KUKA KRL program: ps_res_c2.src, ps_res_c2.dat

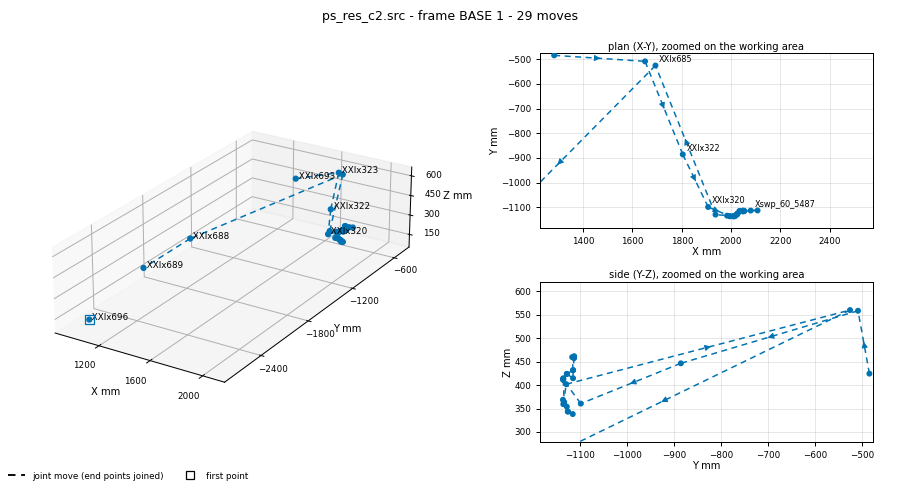
[picture p0: tool path of ps_res_c2.src in frame BASE 1, 29 of 34 moves have a stored position in this frame; points joined in program order, loops and branches not executed]
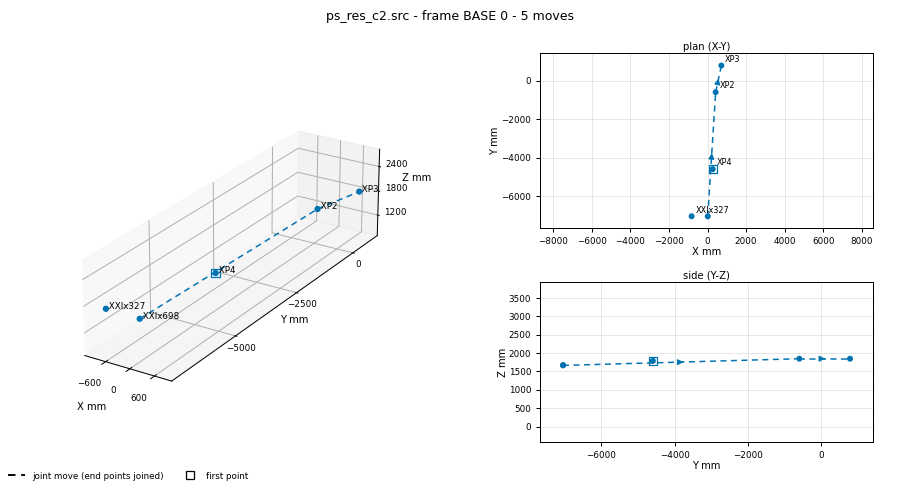
[picture p1: tool path of ps_res_c2.src in frame BASE 0, 5 of 34 moves have a stored position in this frame; points joined in program order, loops and branches not executed]
--- ps_res_c2.src ---
&ACCESS RVO1
&REL 115
&COMMENT Solda GUN C2 respot
&PARAM DISKPATH = KRC:\R1\Program
DEF ps_res_c2( )

;FOLD INI
;FOLD SPOTTECH INI
USERSPOT(#INIT)
;ENDFOLD (SPOTTECH INI)
;FOLD GRIPPERTECH INI
USER_GRP(0,DUMMY,DUMMY,GDEFAULT)
;ENDFOLD (GRIPPERTECH INI)
  ;FOLD USER INI
    ;Make your modifications here

  ;ENDFOLD (USER INI)
;ENDFOLD (INI)

; Caracterização dos meios de produção:
; Versão Atual:
; 08/06/2013 12:00 Name: P13.050-R1 CHANGES: Solda respot Actros
; Gun C2 (F2 6640 0018 997)

chk_w3_wechs_ok ( )              ; CHECK C2

if MaxStandMenge (2) then
 MaxStandmengeErreicht (2)
endif

IF (NOT(GHOST())) THEN
if Elektrodenwechsel (2) then
 e_fraes3 ()
endif
ENDIF

;FOLD OUT 3348 'Fora area GEOBOX' State=FALSE ;%{PE}%R 8.2.20,%MKUKATPBASIS,%COUT,%VOUTX,%P 2:3348, 3:Fora area GEOBOX, 5:FALSE, 6:
$OUT[3348]=FALSE
;ENDFOLD

;FOLD PTP P4 CONT Vel=100 % PDAT40 Tool[3]:GUN C2 Base[0];%{PE}%R 8.2.20,%MKUKATPBASIS,%CMOVE,%VPTP,%P 1:PTP, 2:P4, 3:C_DIS, 5:100, 7:PDAT40
$BWDSTART=FALSE
PDAT_ACT=PPDAT40
FDAT_ACT=FP4
BAS(#PTP_PARAMS,100)
PTP XP4 C_DIS
;ENDFOLD

;FOLD Collision.Monitoring_3_On ;%{PE}%MKUKATPUSER
COLLSTOP( 3, 1 ) ;Interrupt-Controlled
;ENDFOLD

;FOLD PTP Xlx696 CONT Vel=100 % PDAT23 Tool[3]:GUN C2 Base[0];%{PE}%R 8.2.20,%MKUKATPBASIS,%CMOVE,%VPTP,%P 1:PTP, 2:Xlx696, 3:C_DIS, 5:100, 7:PDAT23
$BWDSTART=FALSE
PDAT_ACT=PPDAT23
FDAT_ACT=FXlx696
BAS(#PTP_PARAMS,100)
PTP XXlx696 C_DIS
;ENDFOLD

;FOLD Collision.Monitoring_5_On ;%{PE}%MKUKATPUSER
COLLSTOP( 5, 1 ) ;not Interrupt-Controlled
;ENDFOLD

;FOLD PTP Xlx327 CONT Vel=100 % P_OLP22 Tool[3]:GUN C2 Base[0];%{PE}%R 8.2.20,%MKUKATPBASIS,%CMOVE,%VPTP,%P 1:PTP, 2:Xlx327, 3:C_DIS, 5:100, 7:P_OLP22
$BWDSTART=FALSE
PDAT_ACT=PP_OLP22
FDAT_ACT=FXlx327
BAS(#PTP_PARAMS,100)
PTP XXlx327 C_DIS
;ENDFOLD

;LIGA INTERTRAVAMENTO 15 C/R5
;FOLD Collision.Monitoring_AREA_9_On ;%{PE}%MKUKATPUSER
COLLSTOP( 15, 1 ) ;not Interrupt-Controlled
;ENDFOLD

;FOLD PTP Xlx693 CONT Vel=100 % PDAT20 Tool[3]:GUN C2 Base[0];%{PE}%R 8.2.20,%MKUKATPBASIS,%CMOVE,%VPTP,%P 1:PTP, 2:Xlx693, 3:C_DIS, 5:100, 7:PDAT20
$BWDSTART=FALSE
PDAT_ACT=PPDAT20
FDAT_ACT=FXlx693
BAS(#PTP_PARAMS,100)
PTP XXlx693 C_DIS
;ENDFOLD
;FOLD PTP Xlx323 CONT Vel=100 % P_OLP3 Tool[3]:GUN C2 Base[0];%{PE}%R 8.2.19,%MKUKATPBASIS,%CMOVE,%VPTP,%P 1:PTP, 2:Xlx323, 3:C_DIS, 5:100, 7:P_OLP3
$BWDSTART=FALSE
PDAT_ACT=PP_OLP3
FDAT_ACT=FXlx323
BAS(#PTP_PARAMS,100)
PTP XXlx323 C_DIS
;ENDFOLD
;FOLD PTP Xlx322 CONT Vel=100 % P_OLP4 Tool[3]:GUN C2 Base[0];%{PE}%R 8.2.19,%MKUKATPBASIS,%CMOVE,%VPTP,%P 1:PTP, 2:Xlx322, 3:C_DIS, 5:100, 7:P_OLP4
$BWDSTART=FALSE
PDAT_ACT=PP_OLP4
FDAT_ACT=FXlx322
BAS(#PTP_PARAMS,100)
PTP XXlx322 C_DIS
;ENDFOLD
;FOLD PTP Xlx320 CONT Vel=100 % P_OLP6 Tool[3]:GUN C2 Base[0];%{PE}%R 8.2.19,%MKUKATPBASIS,%CMOVE,%VPTP,%P 1:PTP, 2:Xlx320, 3:C_DIS, 5:100, 7:P_OLP6
$BWDSTART=FALSE
PDAT_ACT=PP_OLP6
FDAT_ACT=FXlx320
BAS(#PTP_PARAMS,100)
PTP XXlx320 C_DIS
;ENDFOLD
;FOLD PTP Xlx669 CONT Vel=100 % PDAT26 Tool[3]:GUN C2 Base[0];%{PE}%R 8.2.20,%MKUKATPBASIS,%CMOVE,%VPTP,%P 1:PTP, 2:Xlx669, 3:C_DIS, 5:100, 7:PDAT26
$BWDSTART=FALSE
PDAT_ACT=PPDAT26
FDAT_ACT=FXlx669
BAS(#PTP_PARAMS,100)
PTP XXlx669 C_DIS
;ENDFOLD
;FOLD PTP Xlx670 CONT Vel=80 % PDAT27 Tool[3]:GUN C2 Base[0];%{PE}%R 8.2.20,%MKUKATPBASIS,%CMOVE,%VPTP,%P 1:PTP, 2:Xlx670, 3:C_DIS, 5:80, 7:PDAT27
$BWDSTART=FALSE
PDAT_ACT=PPDAT27
FDAT_ACT=FXlx670
BAS(#PTP_PARAMS,80)
PTP XXlx670 C_DIS
;ENDFOLD
;FOLD PTP Xlx672 CONT Vel=80 % PDAT7 Tool[3]:GUN C2 Base[0];%{PE}%R 8.2.20,%MKUKATPBASIS,%CMOVE,%VPTP,%P 1:PTP, 2:Xlx672, 3:C_DIS, 5:80, 7:PDAT7
$BWDSTART=FALSE
PDAT_ACT=PPDAT7
FDAT_ACT=FXlx672
BAS(#PTP_PARAMS,80)
PTP XXlx672 C_DIS
;ENDFOLD

;FOLD ; swp_60_5491;%{PE}%R 8.2.20,%MKUKATPBASIS,%CCOMMENT,%VNORMAL,%P 2:swp_60_5491
;ENDFOLD
;FOLD PTP swp_60_5491 P_OLP7 SPOT Gun=2 RETR CLS PgNo1=61 ACTIVE=1 Tool[3]:GUN C2 Base[1]:Actros;%{PE}%R 8.2.2,%MKUKATPSPOT,%CSPOT,%VPTP,%P 1:PTP, 2:swp_60_5491, 3:, 5:100, 7:P_OLP7, 10:2, 12:#FIRST, 14:#CLO, 16:61, 18:1, 20:1, 22:0, 24:1, 25:S_OLP1
$BWDSTART=FALSE
PDAT_ACT=PP_OLP7
FDAT_ACT=Fswp_60_5491
BAS(#PTP_PARAMS,PP_OLP7.VEL)
S_ACT.GUN=2
S_ACT.PAIR=SDEFAULT.PAIR
S_ACT.RETR=#CLO
S_ACT.CLO_TM=1
S_ACT.PGNO1=61
S_ACT.PGNO2=SDEFAULT.PGNO2
S_ACT.PRESS1=SDEFAULT.PRESS1
S_ACT.PRESS2=SDEFAULT.PRESS2
S_READY=FALSE
PTP Xswp_60_5491
USERSPOT(#SPOT, S_ACT)
WAIT FOR S_READY
;ENDFOLD

;FOLD ; swp_60_5489;%{PE}%R 8.2.20,%MKUKATPBASIS,%CCOMMENT,%VNORMAL,%P 2:swp_60_5489
;ENDFOLD
;FOLD PTP swp_60_5489 P_OLP8 SPOT Gun=2 RETR CLS PgNo1=62 ACTIVE=1 Tool[3]:GUN C2 Base[1]:Actros;%{PE}%R 8.2.2,%MKUKATPSPOT,%CSPOT,%VPTP,%P 1:PTP, 2:swp_60_5489, 3:, 5:100, 7:P_OLP8, 10:2, 12:#FIRST, 14:#CLO, 16:62, 18:1, 20:1, 22:0, 24:1, 25:S_OLP2
$BWDSTART=FALSE
PDAT_ACT=PP_OLP8
FDAT_ACT=Fswp_60_5489
BAS(#PTP_PARAMS,PP_OLP8.VEL)
S_ACT.GUN=2
S_ACT.PAIR=SDEFAULT.PAIR
S_ACT.RETR=#CLO
S_ACT.CLO_TM=1
S_ACT.PGNO1=62
S_ACT.PGNO2=SDEFAULT.PGNO2
S_ACT.PRESS1=SDEFAULT.PRESS1
S_ACT.PRESS2=SDEFAULT.PRESS2
S_READY=FALSE
PTP Xswp_60_5489
USERSPOT(#SPOT, S_ACT)
WAIT FOR S_READY
;ENDFOLD

;FOLD PTP Xlx674 CONT Vel=100 % PDAT29 Tool[3]:GUN C2 Base[0];%{PE}%R 8.2.20,%MKUKATPBASIS,%CMOVE,%VPTP,%P 1:PTP, 2:Xlx674, 3:C_DIS, 5:100, 7:PDAT29
$BWDSTART=FALSE
PDAT_ACT=PPDAT29
FDAT_ACT=FXlx674
BAS(#PTP_PARAMS,100)
PTP XXlx674 C_DIS
;ENDFOLD

;FOLD ; swp_60_5487;%{PE}%R 8.2.20,%MKUKATPBASIS,%CCOMMENT,%VNORMAL,%P 2:swp_60_5487
;ENDFOLD
;FOLD PTP swp_60_5487 P_OLP9 SPOT Gun=2 RETR CLS PgNo1=63 ACTIVE=1 Tool[3]:GUN C2 Base[1]:Actros;%{PE}%R 8.2.2,%MKUKATPSPOT,%CSPOT,%VPTP,%P 1:PTP, 2:swp_60_5487, 3:, 5:100, 7:P_OLP9, 10:2, 12:#FIRST, 14:#CLO, 16:63, 18:1, 20:1, 22:0, 24:1, 25:S_OLP3
$BWDSTART=FALSE
PDAT_ACT=PP_OLP9
FDAT_ACT=Fswp_60_5487
BAS(#PTP_PARAMS,PP_OLP9.VEL)
S_ACT.GUN=2
S_ACT.PAIR=SDEFAULT.PAIR
S_ACT.RETR=#CLO
S_ACT.CLO_TM=1
S_ACT.PGNO1=63
S_ACT.PGNO2=SDEFAULT.PGNO2
S_ACT.PRESS1=SDEFAULT.PRESS1
S_ACT.PRESS2=SDEFAULT.PRESS2
S_READY=FALSE
PTP Xswp_60_5487
USERSPOT(#SPOT, S_ACT)
WAIT FOR S_READY
;ENDFOLD

;FOLD ; swp_60_5485;%{PE}%R 8.2.20,%MKUKATPBASIS,%CCOMMENT,%VNORMAL,%P 2:swp_60_5485
;ENDFOLD
;FOLD PTP swp_60_5485 P_OLP10 SPOT Gun=2 RETR CLS PgNo1=64 ACTIVE=1 Tool[3]:GUN C2 Base[1]:Actros;%{PE}%R 8.2.2,%MKUKATPSPOT,%CSPOT,%VPTP,%P 1:PTP, 2:swp_60_5485, 3:, 5:100, 7:P_OLP10, 10:2, 12:#FIRST, 14:#CLO, 16:64, 18:1, 20:1, 22:0, 24:1, 25:S_OLP4
$BWDSTART=FALSE
PDAT_ACT=PP_OLP10
FDAT_ACT=Fswp_60_5485
BAS(#PTP_PARAMS,PP_OLP10.VEL)
S_ACT.GUN=2
S_ACT.PAIR=SDEFAULT.PAIR
S_ACT.RETR=#CLO
S_ACT.CLO_TM=1
S_ACT.PGNO1=64
S_ACT.PGNO2=SDEFAULT.PGNO2
S_ACT.PRESS1=SDEFAULT.PRESS1
S_ACT.PRESS2=SDEFAULT.PRESS2
S_READY=FALSE
PTP Xswp_60_5485
USERSPOT(#SPOT, S_ACT)
WAIT FOR S_READY
;ENDFOLD

;FOLD PTP Xlx328 CONT Vel=100 % PDAT30 Tool[3]:GUN C2 Base[0];%{PE}%R 8.2.20,%MKUKATPBASIS,%CMOVE,%VPTP,%P 1:PTP, 2:Xlx328, 3:C_DIS, 5:100, 7:PDAT30
$BWDSTART=FALSE
PDAT_ACT=PPDAT30
FDAT_ACT=FXlx328
BAS(#PTP_PARAMS,100)
PTP XXlx328 C_DIS
;ENDFOLD
;FOLD PTP Xlx329 CONT Vel=100 % P_OLP12 Tool[3]:GUN C2 Base[0];%{PE}%R 8.2.19,%MKUKATPBASIS,%CMOVE,%VPTP,%P 1:PTP, 2:Xlx329, 3:C_DIS, 5:100, 7:P_OLP12
$BWDSTART=FALSE
PDAT_ACT=PP_OLP12
FDAT_ACT=FXlx329
BAS(#PTP_PARAMS,100)
PTP XXlx329 C_DIS
;ENDFOLD
;FOLD PTP Xlx330 CONT Vel=100 % P_OLP13 Tool[3]:GUN C2 Base[0];%{PE}%R 8.2.19,%MKUKATPBASIS,%CMOVE,%VPTP,%P 1:PTP, 2:Xlx330, 3:C_DIS, 5:100, 7:P_OLP13
$BWDSTART=FALSE
PDAT_ACT=PP_OLP13
FDAT_ACT=FXlx330
BAS(#PTP_PARAMS,100)
PTP XXlx330 C_DIS
;ENDFOLD
;FOLD PTP Xlx675 Vel=80 % PDAT31 Tool[3]:GUN C2 Base[1]:Actros;%{PE}%R 8.2.20,%MKUKATPBASIS,%CMOVE,%VPTP,%P 1:PTP, 2:Xlx675, 3:, 5:80, 7:PDAT31
$BWDSTART=FALSE
PDAT_ACT=PPDAT31
FDAT_ACT=FXlx675
BAS(#PTP_PARAMS,80)
PTP XXlx675
;ENDFOLD
;FOLD PTP Xlx676 CONT Vel=100 % PDAT32 Tool[3]:GUN C2 Base[0];%{PE}%R 8.2.20,%MKUKATPBASIS,%CMOVE,%VPTP,%P 1:PTP, 2:Xlx676, 3:C_DIS, 5:100, 7:PDAT32
$BWDSTART=FALSE
PDAT_ACT=PPDAT32
FDAT_ACT=FXlx676
BAS(#PTP_PARAMS,100)
PTP XXlx676 C_DIS
;ENDFOLD
;FOLD PTP Xlx678 CONT Vel=100 % PDAT33 Tool[3]:GUN C2 Base[0];%{PE}%R 8.2.20,%MKUKATPBASIS,%CMOVE,%VPTP,%P 1:PTP, 2:Xlx678, 3:C_DIS, 5:100, 7:PDAT33
$BWDSTART=FALSE
PDAT_ACT=PPDAT33
FDAT_ACT=FXlx678
BAS(#PTP_PARAMS,100)
PTP XXlx678 C_DIS
;ENDFOLD
;FOLD PTP Xlx679 Vel=80 % PDAT34 Tool[3]:GUN C2 Base[1]:Actros;%{PE}%R 8.2.20,%MKUKATPBASIS,%CMOVE,%VPTP,%P 1:PTP, 2:Xlx679, 3:, 5:80, 7:PDAT34
$BWDSTART=FALSE
PDAT_ACT=PPDAT34
FDAT_ACT=FXlx679
BAS(#PTP_PARAMS,80)
PTP XXlx679
;ENDFOLD
;FOLD PTP Xlx680 CONT Vel=100 % PDAT35 Tool[3]:GUN C2 Base[0];%{PE}%R 8.2.20,%MKUKATPBASIS,%CMOVE,%VPTP,%P 1:PTP, 2:Xlx680, 3:C_DIS, 5:100, 7:PDAT35
$BWDSTART=FALSE
PDAT_ACT=PPDAT35
FDAT_ACT=FXlx680
BAS(#PTP_PARAMS,100)
PTP XXlx680 C_DIS
;ENDFOLD
;FOLD PTP Xlx682 CONT Vel=100 % PDAT10 Tool[3]:GUN C2 Base[0];%{PE}%R 8.2.19,%MKUKATPBASIS,%CMOVE,%VPTP,%P 1:PTP, 2:Xlx682, 3:C_DIS, 5:100, 7:PDAT10
$BWDSTART=FALSE
PDAT_ACT=PPDAT10
FDAT_ACT=FXlx682
BAS(#PTP_PARAMS,100)
PTP XXlx682 C_DIS
;ENDFOLD

;FOLD ; swp_60_5493;%{PE}%R 8.2.20,%MKUKATPBASIS,%CCOMMENT,%VNORMAL,%P 2:swp_60_5493
;ENDFOLD
;FOLD PTP swp_60_5493 P_OLP14 SPOT Gun=2 RETR CLS PgNo1=65 ACTIVE=1 Tool[3]:GUN C2 Base[1]:Actros;%{PE}%R 8.2.2,%MKUKATPSPOT,%CSPOT,%VPTP,%P 1:PTP, 2:swp_60_5493, 3:, 5:100, 7:P_OLP14, 10:2, 12:#FIRST, 14:#CLO, 16:65, 18:1, 20:1, 22:0, 24:1, 25:S_OLP5
$BWDSTART=FALSE
PDAT_ACT=PP_OLP14
FDAT_ACT=Fswp_60_5493
BAS(#PTP_PARAMS,PP_OLP14.VEL)
S_ACT.GUN=2
S_ACT.PAIR=SDEFAULT.PAIR
S_ACT.RETR=#CLO
S_ACT.CLO_TM=1
S_ACT.PGNO1=65
S_ACT.PGNO2=SDEFAULT.PGNO2
S_ACT.PRESS1=SDEFAULT.PRESS1
S_ACT.PRESS2=SDEFAULT.PRESS2
S_READY=FALSE
PTP Xswp_60_5493
USERSPOT(#SPOT, S_ACT)
WAIT FOR S_READY
;ENDFOLD

;FOLD PTP Xlx331 CONT Vel=100 % P_OLP15 Tool[3]:GUN C2 Base[0];%{PE}%R 8.2.19,%MKUKATPBASIS,%CMOVE,%VPTP,%P 1:PTP, 2:Xlx331, 3:C_DIS, 5:100, 7:P_OLP15
$BWDSTART=FALSE
PDAT_ACT=PP_OLP15
FDAT_ACT=FXlx331
BAS(#PTP_PARAMS,100)
PTP XXlx331 C_DIS
;ENDFOLD
;FOLD PTP Xlx332 Vel=80 % P_OLP16 Tool[3]:GUN C2 Base[1]:Actros;%{PE}%R 8.2.20,%MKUKATPBASIS,%CMOVE,%VPTP,%P 1:PTP, 2:Xlx332, 3:, 5:80, 7:P_OLP16
$BWDSTART=FALSE
PDAT_ACT=PP_OLP16
FDAT_ACT=FXlx332
BAS(#PTP_PARAMS,80)
PTP XXlx332
;ENDFOLD
;FOLD PTP Xlx334 CONT Vel=100 % PDAT36 Tool[3]:GUN C2 Base[0];%{PE}%R 8.2.20,%MKUKATPBASIS,%CMOVE,%VPTP,%P 1:PTP, 2:Xlx334, 3:C_DIS, 5:100, 7:PDAT36
$BWDSTART=FALSE
PDAT_ACT=PPDAT36
FDAT_ACT=FXlx334
BAS(#PTP_PARAMS,100)
PTP XXlx334 C_DIS
;ENDFOLD
;FOLD PTP Xlx685 CONT Vel=100 % PDAT12 Tool[3]:GUN C2 Base[0];%{PE}%R 8.2.20,%MKUKATPBASIS,%CMOVE,%VPTP,%P 1:PTP, 2:Xlx685, 3:C_DIS, 5:100, 7:PDAT12
$BWDSTART=FALSE
PDAT_ACT=PPDAT12
FDAT_ACT=FXlx685
BAS(#PTP_PARAMS,100)
PTP XXlx685 C_DIS
;ENDFOLD
;FOLD PTP Xlx688 CONT Vel=100 % PDAT15 Tool[3]:GUN C2 Base[0];%{PE}%R 8.2.19,%MKUKATPBASIS,%CMOVE,%VPTP,%P 1:PTP, 2:Xlx688, 3:C_DIS, 5:100, 7:PDAT15
$BWDSTART=FALSE
PDAT_ACT=PPDAT15
FDAT_ACT=FXlx688
BAS(#PTP_PARAMS,100)
PTP XXlx688 C_DIS
;ENDFOLD
;FOLD PTP Xlx689 Vel=100 % PDAT16 Tool[3]:GUN C2 Base[1]:Actros;%{PE}%R 8.2.20,%MKUKATPBASIS,%CMOVE,%VPTP,%P 1:PTP, 2:Xlx689, 3:, 5:100, 7:PDAT16
$BWDSTART=FALSE
PDAT_ACT=PPDAT16
FDAT_ACT=FXlx689
BAS(#PTP_PARAMS,100)
PTP XXlx689
;ENDFOLD

;FOLD Collision.Monitoring_5_Off . ;%{PE}%MKUKATPUSER
COLLSTOP( 5, 2+0 )
;ENDFOLD

;DESLIGA INTERTRAVAMENTO 15 C/R5
;FOLD Collision.Monitoring_AREA_9_Off . ;%{PE}%MKUKATPUSER
COLLSTOP( 15, 2+0 )
;ENDFOLD

;FOLD PTP Xlx698 Vel=100 % PDAT25 Tool[3]:GUN C2 Base[0];%{PE}%R 8.2.20,%MKUKATPBASIS,%CMOVE,%VPTP,%P 1:PTP, 2:Xlx698, 3:, 5:100, 7:PDAT25
$BWDSTART=FALSE
PDAT_ACT=PPDAT25
FDAT_ACT=FXlx698
BAS(#PTP_PARAMS,100)
PTP XXlx698
;ENDFOLD

;FOLD Collision.Monitoring_3_On ;%{PE}%MKUKATPUSER
COLLSTOP( 3, 1 ) ;Interrupt-Controlled
;ENDFOLD
;FOLD OUT 3348 'Fora area GEOBOX' State=TRUE ;%{PE}%R 8.2.20,%MKUKATPBASIS,%COUT,%VOUTX,%P 2:3348, 3:Fora area GEOBOX, 5:TRUE, 6:
$OUT[3348]=TRUE
;ENDFOLD
;FOLD PULSE 3407 'RESPOT concluido' State=TRUE Time=2 sec;%{PE}%R 8.2.20,%MKUKATPBASIS,%COUT,%VPULSE,%P 2:3407, 3:RESPOT concluido, 5:TRUE, 6:, 8:2
PULSE($OUT[3407], TRUE,2)
;ENDFOLD
end_weld_RESPOT()             ; BIT FIM DE SOLDA RESPOT

;FOLD PTP P2 CONT Vel=100 % PDAT38 Tool[3]:GUN C2 Base[0];%{PE}%R 8.2.20,%MKUKATPBASIS,%CMOVE,%VPTP,%P 1:PTP, 2:P2, 3:C_DIS, 5:100, 7:PDAT38
$BWDSTART=FALSE
PDAT_ACT=PPDAT38
FDAT_ACT=FP2
BAS(#PTP_PARAMS,100)
PTP XP2 C_DIS
;ENDFOLD
;FOLD PTP P3 CONT Vel=100 % PDAT39 Tool[3]:GUN C2 Base[0];%{PE}%R 8.2.20,%MKUKATPBASIS,%CMOVE,%VPTP,%P 1:PTP, 2:P3, 3:C_DIS, 5:100, 7:PDAT39
$BWDSTART=FALSE
PDAT_ACT=PPDAT39
FDAT_ACT=FP3
BAS(#PTP_PARAMS,100)
PTP XP3 C_DIS
;ENDFOLD

IF (NOT(GHOST())) THEN
if FraesAnf (2) then
 e_fraes3 ()
endif
ENDIF

END

--- ps_res_c2.dat ---
&ACCESS RVO1
&REL 115
&COMMENT Solda GUN C2 respot
&PARAM DISKPATH = KRC:\R1\Program
DEFDAT  ps_res_c2
;FOLD EXTERNAL DECLARATIONS;%{PE}%MKUKATPBASIS,%CEXT,%VCOMMON,%P
;FOLD GRIPPERTECH EXT
EXT  H50 (INT  :IN,INT  :IN,INT  :IN,GRP_TYP  :IN )
;ENDFOLD (GRIPPERTECH EXT)
;FOLD SPOTTECH EXT
EXT  USERSPOT (S_COMMAND  :IN,SPOT_TYPE  :IN )
;ENDFOLD (SPOTTECH EXT)
;FOLD BASISTECH EXT;%{PE}%MKUKATPBASIS,%CEXT,%VEXT,%P
EXT  BAS (BAS_COMMAND  :IN,REAL  :IN )
DECL INT SUCCESS
;ENDFOLD (BASISTECH EXT)
;FOLD USER EXT;%{E}%MKUKATPUSER,%CEXT,%VEXT,%P
;Make your modifications here

;ENDFOLD (USER EXT)
;ENDFOLD (EXTERNAL DECLARATIONS)

;# ============ START PATH : swp_p13050r1_l_res_c2 =============
DECL PDAT PP_OLP3={VEL 100.0,ACC 100.0,APO_DIST 100.0,APO_MODE #CDIS}
DECL PDAT PP_OLP4={VEL 100.0,ACC 100.0,APO_DIST 100.0,APO_MODE #CDIS}
DECL PDAT PP_OLP6={VEL 100.0,ACC 100.0,APO_DIST 100.0,APO_MODE #CDIS}
DECL FDAT Fswp_60_5491={TOOL_NO 3,BASE_NO 1,IPO_FRAME #BASE,POINT2[] " "}
DECL PDAT PP_OLP7={VEL 100.0,ACC 100.0,APO_DIST 0.0}
DECL SPOT_TYPE SS_OLP1={GUN 1,PAIR #FIRST,RETR #CLO,CLO_TM 0,PGNO1 1,PRESS1 1.0,PGNO2 0,PRESS2 0.0}
DECL E6POS Xswp_60_5491={X 2034.40295,Y -1115.71399,Z 414.519287,A -0.537424684,B 7.66125584,C -86.3613815,S 2,T 2,E1 -7394.22998,E2 0.0,E3 0.0,E4 0.0,E5 0.0,E6 0.0}
DECL FDAT Fswp_60_5489={TOOL_NO 3,BASE_NO 1,IPO_FRAME #BASE,POINT2[] " "}
DECL PDAT PP_OLP8={VEL 100.0,ACC 100.0,APO_DIST 0.0}
DECL SPOT_TYPE SS_OLP2={GUN 1,PAIR #FIRST,RETR #CLO,CLO_TM 0,PGNO1 1,PRESS1 1.0,PGNO2 0,PRESS2 0.0}
DECL E6POS Xswp_60_5489={X 2053.09009,Y -1115.62305,Z 431.705597,A 0.718700528,B 7.58153105,C -86.2006226,S 2,T 2,E1 -7394.23096,E2 0.0,E3 0.0,E4 0.0,E5 0.0,E6 0.0}
DECL FDAT Fswp_60_5487={TOOL_NO 3,BASE_NO 1,IPO_FRAME #BASE,POINT2[] " "}
DECL PDAT PP_OLP9={VEL 100.0,ACC 100.0,APO_DIST 0.0}
DECL SPOT_TYPE SS_OLP3={GUN 1,PAIR #FIRST,RETR #CLO,CLO_TM 0,PGNO1 1,PRESS1 1.0,PGNO2 0,PRESS2 0.0}
DECL E6POS Xswp_60_5487={X 2079.30493,Y -1113.76294,Z 457.208313,A 0.301905006,B 1.24084997,C -86.230957,S 2,T 2,E1 -7394.229,E2 0.0,E3 0.0,E4 0.0,E5 0.0,E6 0.0}
DECL FDAT Fswp_60_5485={TOOL_NO 3,BASE_NO 1,IPO_FRAME #BASE,POINT2[] " "}
DECL PDAT PP_OLP10={VEL 100.0,ACC 100.0,APO_DIST 0.0}
DECL SPOT_TYPE SS_OLP4={GUN 1,PAIR #FIRST,RETR #CLO,CLO_TM 0,PGNO1 1,PRESS1 1.0,PGNO2 0,PRESS2 0.0}
DECL E6POS Xswp_60_5485={X 2107.21802,Y -1113.31799,Z 461.441193,A 0.0474418513,B -2.6356349,C -86.2260437,S 2,T 2,E1 -7394.22998,E2 0.0,E3 0.0,E4 0.0,E5 0.0,E6 0.0}
DECL PDAT PP_OLP12={VEL 100.0,ACC 100.0,APO_DIST 100.0,APO_MODE #CDIS}
DECL PDAT PP_OLP13={VEL 100.0,ACC 100.0,APO_DIST 100.0,APO_MODE #CDIS}
DECL FDAT Fswp_60_5493={TOOL_NO 3,BASE_NO 1,IPO_FRAME #BASE,POINT2[] " "}
DECL PDAT PP_OLP14={VEL 100.0,ACC 100.0,APO_DIST 0.0}
DECL SPOT_TYPE SS_OLP5={GUN 1,PAIR #FIRST,RETR #CLO,CLO_TM 0,PGNO1 1,PRESS1 1.0,PGNO2 0,PRESS2 0.0}
DECL E6POS Xswp_60_5493={X 2033.578,Y -1116.34204,Z 338.1716,A 1.53081906,B 32.3203697,C -89.8095779,S 2,T 2,E1 -7433.65918,E2 0.0,E3 0.0,E4 0.0,E5 0.0,E6 0.0}
DECL PDAT PP_OLP15={VEL 100.0,ACC 100.0,APO_DIST 100.0,APO_MODE #CDIS}
DECL PDAT PP_OLP16={VEL 100.0,ACC 100.0,APO_DIST 100.0,APO_MODE #CDIS}
DECL BASIS_SUGG_T LAST_BASIS={POINT1[] "P4                      ",POINT2[] "P4                      ",CP_PARAMS[] "CPDAT0                  ",PTP_PARAMS[] "PDAT40                  ",CONT[] "C_DIS                   ",CP_VEL[] "2.0                     ",PTP_VEL[] "100                     ",SYNC_PARAMS[] "SYNCDAT                 ",SPL_NAME[] "S0                      "}
DECL E6POS XXLX323={X 1650.83398,Y -508.477295,Z 558.240723,A 53.8176498,B 15.4406796,C -59.0121613,S 2,T 2,E1 -7240.60498,E2 0.0,E3 0.0,E4 0.0,E5 0.0,E6 0.0}
DECL FDAT FXlx323={TOOL_NO 3,BASE_NO 1,IPO_FRAME #BASE,POINT2[] " ",TQ_STATE FALSE}
DECL E6POS XXLX322={X 1803.87097,Y -885.955627,Z 446.302612,A 22.5301094,B 23.5790291,C -69.1873627,S 2,T 2,E1 -7240.60498,E2 0.0,E3 0.0,E4 0.0,E5 0.0,E6 0.0}
DECL FDAT FXlx322={TOOL_NO 3,BASE_NO 1,IPO_FRAME #BASE,POINT2[] " ",TQ_STATE FALSE}
DECL E6POS XXLX320={X 1906.76404,Y -1099.17297,Z 360.434998,A 1.91697097,B 13.1802101,C -86.8486328,S 2,T 2,E1 -7085.65186,E2 0.0,E3 0.0,E4 0.0,E5 0.0,E6 0.0}
DECL FDAT FXlx320={TOOL_NO 3,BASE_NO 1,IPO_FRAME #BASE,POINT2[] " ",TQ_STATE FALSE}
DECL E6POS XXLX669={X 1995.33203,Y -1136.65405,Z 411.277893,A -5.59488201,B 13.8034401,C -88.8874893,S 2,T 2,E1 -7181.55615,E2 0.0,E3 0.0,E4 0.0,E5 0.0,E6 0.0}
DECL FDAT FXlx669={TOOL_NO 3,BASE_NO 1,IPO_FRAME #BASE,POINT2[] " ",TQ_STATE FALSE}
DECL E6POS XXLX670={X 2010.49902,Y -1136.55103,Z 413.941406,A -5.59851694,B 13.8267899,C -88.9180527,S 2,T 2,E1 -7181.57324,E2 0.0,E3 0.0,E4 0.0,E5 0.0,E6 0.0}
DECL FDAT FXlx670={TOOL_NO 3,BASE_NO 1,IPO_FRAME #BASE,POINT2[] " ",TQ_STATE FALSE}
DECL E6POS XXLX672={X 2023.67297,Y -1128.95496,Z 423.68399,A 1.14589405,B 7.52097511,C -85.9493637,S 2,T 2,E1 -7393.78711,E2 0.0,E3 0.0,E4 0.0,E5 0.0,E6 0.0}
DECL FDAT FXlx672={TOOL_NO 3,BASE_NO 1,IPO_FRAME #BASE,POINT2[] " ",TQ_STATE FALSE}
DECL PDAT PPDAT7={VEL 100.0,ACC 100.0,APO_DIST 100.0,APO_MODE #CDIS}
DECL E6POS XXLX674={X 2047.89001,Y -1117.51099,Z 459.454102,A 0.300933689,B 1.24180603,C -86.2282486,S 2,T 2,E1 -7394.22998,E2 0.0,E3 0.0,E4 0.0,E5 0.0,E6 0.0}
DECL FDAT FXlx674={TOOL_NO 3,BASE_NO 1,IPO_FRAME #BASE,POINT2[] " ",TQ_STATE FALSE}
DECL E6POS XXLX328={X 2048.87598,Y -1113.43799,Z 458.731201,A 0.0438987799,B -2.63536,C -86.2242966,S 2,T 2,E1 -7394.229,E2 0.0,E3 0.0,E4 0.0,E5 0.0,E6 0.0}
DECL FDAT FXlx328={TOOL_NO 3,BASE_NO 1,IPO_FRAME #BASE,POINT2[] " ",TQ_STATE FALSE}
DECL E6POS XXLX329={X 2053.08496,Y -1115.63403,Z 431.73291,A 0.718055904,B 7.57939482,C -86.1996918,S 2,T 2,E1 -7394.23096,E2 0.0,E3 0.0,E4 0.0,E5 0.0,E6 0.0}
DECL FDAT FXlx329={TOOL_NO 3,BASE_NO 1,IPO_FRAME #BASE,POINT2[] " ",TQ_STATE FALSE}
DECL E6POS XXLX330={X 2023.672,Y -1128.95496,Z 423.685211,A 1.14586604,B 7.52080584,C -85.9492264,S 2,T 2,E1 -7393.78711,E2 0.0,E3 0.0,E4 0.0,E5 0.0,E6 0.0}
DECL FDAT FXlx330={TOOL_NO 3,BASE_NO 1,IPO_FRAME #BASE,POINT2[] " ",TQ_STATE FALSE}
DECL E6POS XXLX675={X 2010.49695,Y -1136.55396,Z 413.941406,A -5.59872198,B 13.8268003,C -88.9183197,S 2,T 2,E1 -7181.57324,E2 0.0,E3 0.0,E4 0.0,E5 0.0,E6 0.0}
DECL FDAT FXlx675={TOOL_NO 3,BASE_NO 1,IPO_FRAME #BASE,POINT2[] " ",TQ_STATE FALSE}
DECL E6POS XXLX676={X 1995.32996,Y -1136.65601,Z 411.270905,A -5.59505701,B 13.8035603,C -88.8872833,S 2,T 2,E1 -7181.55615,E2 0.0,E3 0.0,E4 0.0,E5 0.0,E6 0.0}
DECL FDAT FXlx676={TOOL_NO 3,BASE_NO 1,IPO_FRAME #BASE,POINT2[] " ",TQ_STATE FALSE}
DECL E6POS XXLX678={X 1983.73999,Y -1134.49805,Z 363.461914,A -5.45675516,B 20.0822392,C -88.8476715,S 2,T 2,E1 -7433.646,E2 0.0,E3 0.0,E4 0.0,E5 0.0,E6 0.0}
DECL FDAT FXlx678={TOOL_NO 3,BASE_NO 1,IPO_FRAME #BASE,POINT2[] " ",TQ_STATE FALSE}
DECL E6POS XXLX679={X 2008.52795,Y -1137.172,Z 368.483612,A -3.9182539,B 19.7608109,C -91.7341614,S 2,T 2,E1 -7433.64795,E2 0.0,E3 0.0,E4 0.0,E5 0.0,E6 0.0}
DECL FDAT FXlx679={TOOL_NO 3,BASE_NO 1,IPO_FRAME #BASE,POINT2[] " ",TQ_STATE FALSE}
DECL E6POS XXLX680={X 2023.79102,Y -1129.03503,Z 354.003387,A -1.84301496,B 19.5065002,C -91.6574402,S 2,T 2,E1 -7433.646,E2 0.0,E3 0.0,E4 0.0,E5 0.0,E6 0.0}
DECL FDAT FXlx680={TOOL_NO 3,BASE_NO 1,IPO_FRAME #BASE,POINT2[] " ",TQ_STATE FALSE}
DECL E6POS XXLX682={X 2025.74097,Y -1126.81799,Z 343.535614,A -2.14617491,B 28.6473293,C -91.7823563,S 2,T 2,E1 -7433.64795,E2 0.0,E3 0.0,E4 0.0,E5 0.0,E6 0.0}
DECL FDAT FXlx682={TOOL_NO 3,BASE_NO 1,IPO_FRAME #BASE,POINT2[] " ",TQ_STATE FALSE}
DECL PDAT PPDAT10={VEL 100.0,ACC 100.0,APO_DIST 100.0,APO_MODE #CDIS}
DECL E6POS XXLX331={X 2025.74097,Y -1126.81799,Z 343.535614,A -2.14617491,B 28.6473293,C -91.7823563,S 2,T 2,E1 -7433.64795,E2 0.0,E3 0.0,E4 0.0,E5 0.0,E6 0.0}
DECL FDAT FXlx331={TOOL_NO 3,BASE_NO 1,IPO_FRAME #BASE,POINT2[] " ",TQ_STATE FALSE}
DECL E6POS XXLX332={X 2015.82703,Y -1136.47595,Z 359.285492,A -5.7835288,B 28.0421295,C -93.5095825,S 2,T 2,E1 -7433.65088,E2 0.0,E3 0.0,E4 0.0,E5 0.0,E6 0.0}
DECL FDAT FXlx332={TOOL_NO 3,BASE_NO 1,IPO_FRAME #BASE,POINT2[] " ",TQ_STATE FALSE}
DECL E6POS XXLX334={X 1936.66699,Y -1130.13098,Z 401.784698,A -5.77895784,B 28.0355301,C -93.504097,S 2,T 2,E1 -7433.64697,E2 0.0,E3 0.0,E4 0.0,E5 0.0,E6 0.0}
DECL FDAT FXlx334={TOOL_NO 3,BASE_NO 1,IPO_FRAME #BASE,POINT2[] " ",TQ_STATE FALSE}
DECL E6POS XXLX685={X 1693.04602,Y -525.445679,Z 559.736877,A 52.718399,B 15.4406605,C -59.0119514,S 2,T 2,E1 -7240.60498,E2 0.0,E3 0.0,E4 0.0,E5 0.0,E6 0.0}
DECL FDAT FXlx685={TOOL_NO 3,BASE_NO 1,IPO_FRAME #BASE,POINT2[] " ",TQ_STATE FALSE}
DECL PDAT PPDAT12={VEL 100.0,ACC 100.0,APO_DIST 100.0,APO_MODE #CDIS}
DECL E6POS XXLX688={X 912.772827,Y -1314.802,Z 175.730499,A 93.0003433,B 39.3733711,C 1.569556,S 2,T 2,E1 -5917.896,E2 0.0,E3 0.0,E4 0.0,E5 0.0,E6 0.0}
DECL FDAT FXlx688={TOOL_NO 3,BASE_NO 1,IPO_FRAME #BASE,POINT2[] " ",TQ_STATE FALSE}
DECL PDAT PPDAT15={VEL 100.0,ACC 100.0,APO_DIST 100.0,APO_MODE #CDIS}
DECL E6POS XXLX689={X 904.760681,Y -1887.92297,Z 167.833206,A 93.0698624,B 39.3455315,C 1.46217704,S 2,T 2,E1 -5915.4541,E2 0.0,E3 0.0,E4 0.0,E5 0.0,E6 0.0}
DECL FDAT FXlx689={TOOL_NO 3,BASE_NO 1,IPO_FRAME #BASE,POINT2[] " ",TQ_STATE FALSE}
DECL PDAT PPDAT16={VEL 100.0,ACC 100.0,APO_DIST 100.0,APO_MODE #CDIS}
DECL SPOT_SUGG_T LAST_SPOT={GUN[] " 1                      ",RETR_CMD[] "#OPN                    ",CHOISE[] "#FIRST                  ",CLO_TM[] "0                       ",PGNO1[] " 1                      ",PRESS1[] "0                       ",PGNO2[] " 1                      ",PRESS2[] "0                       ",SPOT_PARAMS[] "NORMAL                  "}
DECL E6POS XXLX693={X 1282.38501,Y -484.164307,Z 424.302399,A 87.946907,B 37.2855606,C -72.154892,S 2,T 2,E1 -5924.74316,E2 0.0,E3 0.0,E4 0.0,E5 0.0,E6 0.0}
DECL FDAT FXlx693={TOOL_NO 3,BASE_NO 1,IPO_FRAME #BASE,POINT2[] " ",TQ_STATE FALSE}
DECL PDAT PPDAT20={VEL 100.0,ACC 100.0,APO_DIST 50.0,APO_MODE #CDIS}
DECL PDAT PP_OLP22={VEL 100.0,ACC 100.0,APO_DIST 100.0,APO_MODE #CDIS}
DECL E6POS XXlx327={X -825.171814,Y -7036.83398,Z 1674.80103,A 175.981201,B 39.6716003,C -9.74450207,S 2,T 2,E1 -5583.99609,E2 0.0,E3 0.0,E4 0.0,E5 0.0,E6 0.0}
DECL FDAT FXlx327={TOOL_NO 3,BASE_NO 0,IPO_FRAME #BASE,POINT2[] " ",TQ_STATE FALSE}
DECL PDAT PPDAT23={VEL 100.0,ACC 100.0,APO_DIST 100.0,APO_MODE #CDIS}
DECL E6POS XXlx696={X 1051.505,Y -2731.65698,Z 159.500198,A 158.389099,B 88.6550827,C 158.968201,S 2,T 2,E1 -5289.49219,E2 0.0,E3 0.0,E4 0.0,E5 0.0,E6 0.0}
DECL FDAT FXlx696={TOOL_NO 3,BASE_NO 1,IPO_FRAME #BASE,POINT2[] " ",TQ_STATE FALSE}
DECL PDAT PPDAT25={VEL 100.0,ACC 100.0,APO_DIST 100.0,APO_MODE #CDIS}
DECL E6POS XXlx698={X 11.6570301,Y -7041.73389,Z 1665.0,A -111.610901,B 88.6550827,C 158.968201,S 2,T 2,E1 -5289.49219,E2 0.0,E3 0.0,E4 0.0,E5 0.0,E6 0.0}
DECL FDAT FXlx698={TOOL_NO 3,BASE_NO 0,IPO_FRAME #BASE,POINT2[] " ",TQ_STATE FALSE}
DECL PDAT PPDAT26={VEL 100.0,ACC 100.0,APO_DIST 10.0,APO_MODE #CDIS}
DECL PDAT PPDAT27={VEL 100.0,ACC 100.0,APO_DIST 10.0,APO_MODE #CDIS}
DECL PDAT PPDAT29={VEL 100.0,ACC 100.0,APO_DIST 10.0,APO_MODE #CDIS}
DECL PDAT PPDAT30={VEL 100.0,ACC 100.0,APO_DIST 10.0,APO_MODE #CDIS}
DECL PDAT PPDAT31={VEL 100.0,ACC 100.0,APO_DIST 10.0,APO_MODE #CDIS}
DECL PDAT PPDAT32={VEL 100.0,ACC 100.0,APO_DIST 10.0,APO_MODE #CDIS}
DECL PDAT PPDAT33={VEL 100.0,ACC 100.0,APO_DIST 10.0,APO_MODE #CDIS}
DECL PDAT PPDAT34={VEL 100.0,ACC 100.0,APO_DIST 10.0,APO_MODE #CDIS}
DECL PDAT PPDAT35={VEL 100.0,ACC 100.0,APO_DIST 10.0,APO_MODE #CDIS}
DECL PDAT PPDAT36={VEL 100.0,ACC 100.0,APO_DIST 10.0,APO_MODE #CDIS}
DECL PDAT PPDAT38={VEL 100.0,ACC 100.0,APO_DIST 100.0,APO_MODE #CDIS}
DECL E6POS XP2={X 421.536194,Y -599.552307,Z 1847.63794,A -94.9410782,B 80.8796997,C 79.033371,S 2,T 2,E1 213.667007,E2 0.0,E3 0.0,E4 0.0,E5 0.0,E6 0.0}
DECL FDAT FP2={TOOL_NO 3,BASE_NO 0,IPO_FRAME #BASE,POINT2[] " ",TQ_STATE FALSE}
DECL PDAT PPDAT39={VEL 100.0,ACC 100.0,APO_DIST 100.0,APO_MODE #CDIS}
DECL E6POS XP3={X 718.102417,Y 782.301575,Z 1847.63904,A 6.03337288,B 80.8794937,C 79.033287,S 2,T 3,E1 213.666397,E2 0.0,E3 0.0,E4 0.0,E5 0.0,E6 0.0}
DECL FDAT FP3={TOOL_NO 3,BASE_NO 0,IPO_FRAME #BASE,POINT2[] " ",TQ_STATE FALSE}
DECL E6POS XP4={X 269.370514,Y -4591.70801,Z 1791.08704,A -98.3080826,B 85.59655,C 133.9263,S 2,T 2,E1 -3107.69409,E2 0.0,E3 0.0,E4 0.0,E5 0.0,E6 0.0}
DECL FDAT FP4={TOOL_NO 3,BASE_NO 0,IPO_FRAME #BASE,POINT2[] " ",TQ_STATE FALSE}
DECL PDAT PPDAT40={VEL 100.0,ACC 100.0,APO_DIST 100.0,APO_MODE #CDIS}
ENDDAT
